Fanuc KAREL source: kt00901.KL

-- PROVISIONAL review KL for V940-1; original PC SHA256 dabe46131533726eb3a4b370479b166b7708cb3cb1da2838068ea46dbb894591
-- Incomplete behavior may be omitted. Consult companion uncertainty JSON. Do not deploy.
PROGRAM KT00901
%NOLOCKGROUP
VAR
  OUT : BOOLEAN
-- UNRESOLVED_DECL P1 type=000199
-- UNRESOLVED_DECL P2 type=000199
BEGIN
  -- V9_ZERO_TABLE_METADATA_HINT layout=0001; no indexed target words; source/name/runtime held
  -- UNRESOLVED_PC offsets 5-28; opcodes 27,22,1C,27,9D,76,23
  -- UNRESOLVED_PC offsets 33-37; opcodes 7F
END KT00901
